FUNCTION_BLOCK ABSTRACT BaseCylinder IMPLEMENTS ITF_Cylinder
VAR_INPUT
END_VAR
VAR_OUTPUT
END_VAR
VAR
	//Hardware
	DI_Extended AT %I* : BOOL;
	DI_Retracted AT %I* : BOOL;
	DO_Extend AT %Q* : BOOL;
	//NOT USED BUT USABLE	
	DI_BoundaryPressure AT %I* : BOOL;
	DI_BoundaryFlowPressure AT %I* : BOOL;
	AI_PressureSensor AT %I* : INT;
	AI_FlowPressure AT %I* : INT;
	AI_PositionTransmitter AT %I* : INT;
END_VAR

PROPERTY Extended : BOOL
GET
Extended := DI_Extended;
END_GET
END_PROPERTY

METHOD ABSTRACT METH_Extend : BOOL
END_METHOD

METHOD ABSTRACT METH_Retract : BOOL
END_METHOD

PROPERTY Retracted : BOOL
GET
Retracted := DI_Retracted;
END_GET
END_PROPERTY

END_FUNCTION_BLOCK

(* stored: Version 1.1.0.1
   POU BaseCylinder: Id {36b2f985-d5f3-48e5-b80f-dac311c9bd0d}, SpecialFunc None
   Property Extended: Id {9367427e-a835-4ef4-b154-d791f37f3f22}
   Get Get: Id {2817200b-01a6-4881-8fcb-9b4d452386df}
   Method METH_Extend: Id {5e0ba800-5d79-4df2-a234-753f93e95d9d}
   Method METH_Retract: Id {6f018710-d838-4c74-b33d-83bb4eeb23f1}
   Property Retracted: Id {94a5ad90-698f-486b-b4d1-4bb9819771f8}
   Get Get: Id {efbc6477-e169-400e-a903-88ef8cb38647} *)
